// TIA Portal V17 export
// export: Created 2022-07-20T06:59:50.7131062Z, ExportSetting WithDefaults, DisplayName Totally Integrated Automation Portal, DisplayVersion V17, DisplayName TIA Portal Openness, DisplayVersion V17, DisplayName TIA Portal Version Control Interface, DisplayVersion V17, DisplayName SINAMICS Startdrive Advanced, DisplayVersion V17, DisplayName SINAMICS Startdrive G130, G150, S120, S150, SINAMICS MV, S210, DisplayVersion V17, DisplayName SINAMICS Startdrive G110M, G120, G120C, G120D, G120P, G115D, DisplayVersion V17, DisplayName STEP 7 Professional, DisplayVersion V17, DisplayName STEP 7 Safety, DisplayVersion V17, DisplayName WinCC Advanced, DisplayVersion V17
FUNCTION_BLOCK "FB10062_IperPrintingHeadsTray"   // FB10062, LAD
{ S7_Optimized_Access := 'TRUE' }
VERSION : 0.1
// stored: AutoNumber false, IsIECCheckEnabled false, IsRetainMemResEnabled false, MemoryReserve 100, SetENOAutomatically false, UDAEnableTagReadback false
   VAR_INPUT
      ToAxis : TO_PositioningAxis;
      HomingSensor : Bool;
      RequestHoming : Bool;
      RequestGoToClearancePosition : Bool;
      RequestGoToCleaningPosition : Bool;
      RequestGoToCappingStationPosition : Bool;
      RequestGoToWipingPosition : Bool;
      RequestGoToWipePosition : Bool;
      RequestGoToPurgePosition : Bool;
      RequestGoToUnjamPosition : Bool;
      RequestGoToPrintPosition : Bool;
      RequestStopMotor : Bool;
      RequestAcknowledge : Bool;
      ClearancePosition : LReal;
      CleaningPosition : LReal;
      CappingStationPosition : LReal;
      WipingPosition : LReal;
      WipePosition : LReal;
      PurgePosition : LReal;
      StandByPosition : LReal;
      PrintPosition : LReal;
   END_VAR
   VAR_OUTPUT
      AxisPositionningTooLong : Bool;
      HomingDone : Bool;
      ActualPosition_mm : LReal;
      IsInClearancePosition : Bool;
      IsInCleaningPosition : Bool;
      IsInCappingStationPosition : Bool;
      IsInWipingPosition : Bool;
      IsInWipePosition : Bool;
      IsInPurgePosition : Bool;
      IsInUnjamPosition : Bool;
      IsInPrintPosition : Bool;
   END_VAR
   VAR_IN_OUT
      AxisStructure : "LAxisCtrl_Pos";
   END_VAR
   VAR
      FB10400_APCMotor_Instance { S7_SetPoint := 'True'} : "FB10400_APCMotor";
      test { S7_SetPoint := 'True'} : LReal;
   END_VAR
BEGIN

REGION Network 1 (SCL): First Scan
   IF "FirstScan" THEN
       #HomingDone := FALSE;
       #IsInClearancePosition := FALSE;
       #IsInCleaningPosition := FALSE;
       #IsInCappingStationPosition := FALSE;
       #IsInWipingPosition := FALSE;
       #IsInWipePosition := FALSE;
       #IsInPurgePosition := FALSE;
       #IsInUnjamPosition := FALSE;
       #IsInPrintPosition := FALSE;
   END_IF;
END_REGION

REGION Network 2: Printing System 1 Heads Tray Management
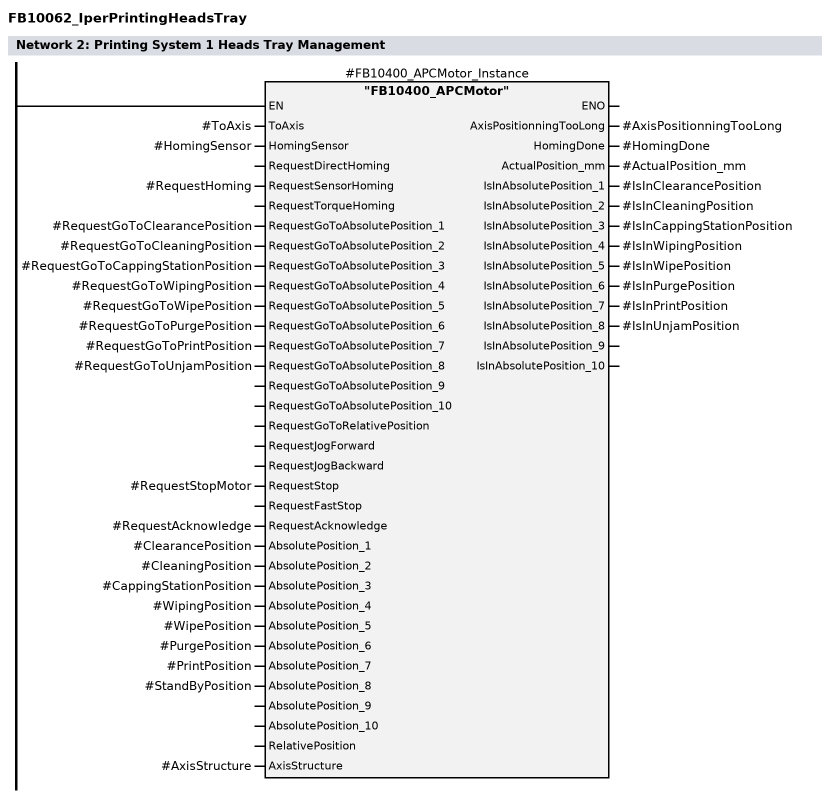
   RUNG wire#powerrail
      #FB10400_APCMotor_Instance(ToAxis := #ToAxis, HomingSensor := #HomingSensor, RequestDirectHoming :=, RequestSensorHoming := #RequestHoming, RequestTorqueHoming :=, RequestGoToAbsolutePosition_1 := #RequestGoToClearancePosition, RequestGoToAbsolutePosition_2 := #RequestGoToCleaningPosition, RequestGoToAbsolutePosition_3 := #RequestGoToCappingStationPosition, RequestGoToAbsolutePosition_4 := #RequestGoToWipingPosition, RequestGoToAbsolutePosition_5 := #RequestGoToWipePosition, RequestGoToAbsolutePosition_6 := #RequestGoToPurgePosition, RequestGoToAbsolutePosition_7 := #RequestGoToPrintPosition, RequestGoToAbsolutePosition_8 := #RequestGoToUnjamPosition, RequestGoToAbsolutePosition_9 :=, RequestGoToAbsolutePosition_10 :=, RequestGoToRelativePosition :=, RequestJogForward :=, RequestJogBackward :=, RequestStop := #RequestStopMotor, RequestFastStop :=, RequestAcknowledge := #RequestAcknowledge, AbsolutePosition_1 := #ClearancePosition, AbsolutePosition_2 := #CleaningPosition, AbsolutePosition_3 := #CappingStationPosition, AbsolutePosition_4 := #WipingPosition, AbsolutePosition_5 := #WipePosition, AbsolutePosition_6 := #PurgePosition, AbsolutePosition_7 := #PrintPosition, AbsolutePosition_8 := #StandByPosition, AbsolutePosition_9 :=, AbsolutePosition_10 :=, RelativePosition :=, AxisStructure := #AxisStructure, AxisPositionningTooLong => #AxisPositionningTooLong, HomingDone => #HomingDone, ActualPosition_mm => #ActualPosition_mm, IsInAbsolutePosition_1 => #IsInClearancePosition, IsInAbsolutePosition_2 => #IsInCleaningPosition, IsInAbsolutePosition_3 => #IsInCappingStationPosition, IsInAbsolutePosition_4 => #IsInWipingPosition, IsInAbsolutePosition_5 => #IsInWipePosition, IsInAbsolutePosition_6 => #IsInPurgePosition, IsInAbsolutePosition_7 => #IsInPrintPosition, IsInAbsolutePosition_8 => #IsInUnjamPosition, IsInAbsolutePosition_9 =>, IsInAbsolutePosition_10 =>)
   END_RUNG
   // the same network as SCL:
   #FB10400_APCMotor_Instance(ToAxis := #ToAxis,   // "FB10400_APCMotor"
                           HomingSensor := #HomingSensor,
                           RequestSensorHoming := #RequestHoming,
                           RequestGoToAbsolutePosition_1 := #RequestGoToClearancePosition,
                           RequestGoToAbsolutePosition_2 := #RequestGoToCleaningPosition,
                           RequestGoToAbsolutePosition_3 := #RequestGoToCappingStationPosition,
                           RequestGoToAbsolutePosition_4 := #RequestGoToWipingPosition,
                           RequestGoToAbsolutePosition_5 := #RequestGoToWipePosition,
                           RequestGoToAbsolutePosition_6 := #RequestGoToPurgePosition,
                           RequestGoToAbsolutePosition_7 := #RequestGoToPrintPosition,
                           RequestGoToAbsolutePosition_8 := #RequestGoToUnjamPosition,
                           RequestStop := #RequestStopMotor,
                           RequestAcknowledge := #RequestAcknowledge,
                           AbsolutePosition_1 := #ClearancePosition,
                           AbsolutePosition_2 := #CleaningPosition,
                           AbsolutePosition_3 := #CappingStationPosition,
                           AbsolutePosition_4 := #WipingPosition,
                           AbsolutePosition_5 := #WipePosition,
                           AbsolutePosition_6 := #PurgePosition,
                           AbsolutePosition_7 := #PrintPosition,
                           AbsolutePosition_8 := #StandByPosition,
                           AxisStructure := #AxisStructure,
                           AxisPositionningTooLong => #AxisPositionningTooLong,
                           HomingDone => #HomingDone,
                           ActualPosition_mm => #ActualPosition_mm,
                           IsInAbsolutePosition_1 => #IsInClearancePosition,
                           IsInAbsolutePosition_2 => #IsInCleaningPosition,
                           IsInAbsolutePosition_3 => #IsInCappingStationPosition,
                           IsInAbsolutePosition_4 => #IsInWipingPosition,
                           IsInAbsolutePosition_5 => #IsInWipePosition,
                           IsInAbsolutePosition_6 => #IsInPurgePosition,
                           IsInAbsolutePosition_7 => #IsInPrintPosition,
                           IsInAbsolutePosition_8 => #IsInUnjamPosition);
END_REGION
END_FUNCTION_BLOCK
